FUNCTION_BLOCK FB_ChangeTrig
VAR_INPUT
END_VAR
VAR_OUTPUT
END_VAR
VAR
	internalPointer:POINTER TO BYTE;
	aBytes:ARRAY[0..254] OF BYTE;
END_VAR

METHOD M_ChngTrig : BOOL
VAR_INPUT
	in:ANY;
END_VAR
IF THIS^.internalPointer <> 0 THEN
	M_ChngTrig:= memcmp(in.pValue,THIS^.internalPointer, in.diSize) <> 0;
	memcpy(THIS^.internalPointer,in.pValue,in.diSize);
ELSE
	THIS^.internalPointer:= ADR(THIS^.aBytes);
END_IF
END_METHOD

END_FUNCTION_BLOCK

(* stored: Version 1.1.0.1, ProductVersion 3.1.4024.11
   POU FB_ChangeTrig: Id {bbc9f587-9e81-40a3-9d13-3a200d8f7b93}, SpecialFunc None
   Method M_ChngTrig: Id {d075d354-de21-4567-9805-9b120eace341} *)
